(* PLC project Example1, KAIST_SELAB noNameNow 1.0 *)
(* stored: creationDateTime 2019-01-14T15:39:07, modificationDateTime 2019-03-13T12:08:51 *)

PROGRAM program0
  VAR_IN_OUT
    CTU_UP : BOOL;
  END_VAR
  VAR_INPUT
    FILL_BIN : BOOL;
    PULSE_TIME : INT;
    BIN_EMPTY : BOOL;
    SETPOINT : INT;
  END_VAR
  VAR_OUTPUT
    TON_et : INT;
    BIN_LEVEL : INT;
    CTU_Q : BOOL;
  END_VAR
  VAR
    PULSE : TON;
    LEVEL_CTR : CTU;
  END_VAR
  VAR  (* added by the conversion: wires and edge detectors of the diagram *)
    R_TRIG1 : R_TRIG;
  END_VAR

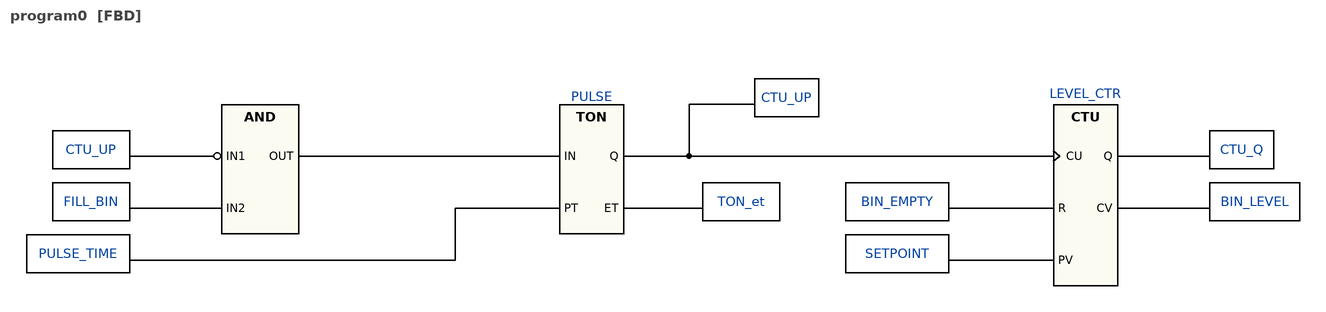
(* FBD diagram, written out as Structured Text *)
PULSE(IN := NOT CTU_UP AND FILL_BIN, PT := PULSE_TIME);
CTU_UP := PULSE.Q;
R_TRIG1(CLK := PULSE.Q);
LEVEL_CTR(CU := R_TRIG1.Q, R := BIN_EMPTY, PV := SETPOINT);
CTU_Q := LEVEL_CTR.Q;
TON_et := PULSE.ET;
BIN_LEVEL := LEVEL_CTR.CV;
END_PROGRAM
